SUBAPPLICATION MSG_PUBLISHER (* ROS 2 MSG Publisher *)
  (* Standard: 61499-2 *)
  (* Version 1.0, 2023-03-14, Tim Hesse *)
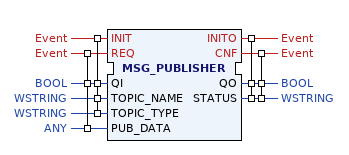
  EVENT_INPUT
    INIT WITH QI, TOPIC_NAME, TOPIC_TYPE; (* Initialization Request *)
    REQ WITH QI, PUB_DATA; (* Normal Execution Request *)
  END_EVENT
  EVENT_OUTPUT
    INITO WITH QO, STATUS; (* Initialization Confirm *)
    CNF WITH QO, STATUS; (* Execution Confirmation *)
  END_EVENT
  VAR_INPUT
    QI : BOOL; (* Input event qualifier *)
    TOPIC_NAME : WSTRING; (* ROS 2 Topic Name *)
    TOPIC_TYPE : WSTRING; (* ROS 2 Topic Type *)
    PUB_DATA : ANY; (* Data to publish *)
  END_VAR
  VAR_OUTPUT
    QO : BOOL; (* Output event qualifier *)
    STATUS : WSTRING; (* Service Status *)
  END_VAR
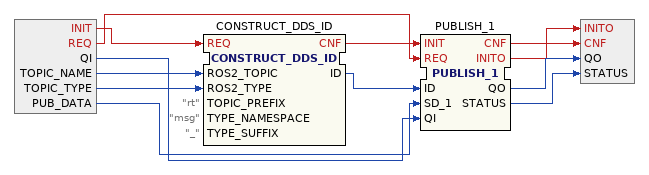
  FBS
    CONSTRUCT_DDS_ID : CONSTRUCT_DDS_ID(TOPIC_PREFIX := "rt", TYPE_NAMESPACE := "msg", TYPE_SUFFIX := "_");
    PUBLISH_1 : PUBLISH_1;
  END_FBS
  EVENT_CONNECTIONS
    INIT TO CONSTRUCT_DDS_ID.REQ;
    CONSTRUCT_DDS_ID.CNF TO PUBLISH_1.INIT;
    PUBLISH_1.CNF TO CNF;
    PUBLISH_1.INITO TO INITO;
    REQ TO PUBLISH_1.REQ;
  END_CONNECTIONS
  DATA_CONNECTIONS
    CONSTRUCT_DDS_ID.ID TO PUBLISH_1.ID;
    TOPIC_NAME TO CONSTRUCT_DDS_ID.ROS2_TOPIC;
    TOPIC_TYPE TO CONSTRUCT_DDS_ID.ROS2_TYPE;
    PUB_DATA TO PUBLISH_1.SD_1;
    QI TO PUBLISH_1.QI;
    PUBLISH_1.QO TO QO;
    PUBLISH_1.STATUS TO STATUS;
  END_CONNECTIONS
END_SUBAPPLICATION
